Staubli VAL3: calc_WinningNumber.pgx

program calc_WinningNumber(num& x_nCurrentMatrix[] (dimensions=2), num x_nCurrentNumber, num& x_nRESULT)
  local num l_nX
  local num l_nY
begin

  //resize(x_nRESULT,1,1)
  x_nRESULT = 0
  for l_nX = 0 to size(x_nCurrentMatrix,1)-1
    for l_nY = 0 to size(x_nCurrentMatrix,2)-1
      x_nRESULT = x_nRESULT + x_nCurrentMatrix[l_nX, l_nY]
    endFor
  endFor

  x_nRESULT = x_nRESULT*x_nCurrentNumber

end
